FUNCTION_BLOCK FB_SimulatedPump EXTENDS FB_ComponentBase IMPLEMENTS I_Pump
VAR_INPUT
END_VAR
VAR_OUTPUT
END_VAR
VAR
END_VAR

{warning 'Add method implementation '}
METHOD CyclicLogic
END_METHOD

{warning 'Add property implementation'}
PROPERTY Speed : LREAL
GET
END_GET
SET
END_SET
END_PROPERTY

{warning 'Add method implementation '}
METHOD Start : BOOL
END_METHOD

{warning 'Add method implementation '}
METHOD Stop
END_METHOD

END_FUNCTION_BLOCK

(* stored: Version 1.1.0.1
   POU FB_SimulatedPump: Id {be317f72-b581-4b21-abf7-8ef72808cd18}, SpecialFunc None
   Method CyclicLogic: Id {0714ccf9-99b3-4d76-bd27-1f6e735a0fba}
   Property Speed: Id {ed4b2892-e48c-40a5-9f09-396963c2d4bf}
   Get Get: Id {5da42a9b-3caa-479a-bbc2-6ba02383d132}
   Set Set: Id {c134a5e9-7506-45c1-8311-f133b1759a3f}
   Method Start: Id {f9ac44a6-3592-47b1-a865-0211ed52e8d7}
   Method Stop: Id {a18011b8-543a-48c9-9242-affb8168b7ff} *)
